// Mitsubishi GX Works2 project: timer   PLC: Q03UDV

PROGRAM MAIN
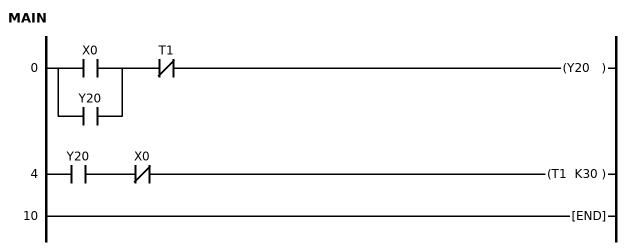
0     LD      X0
      OR      Y20
      ANI     T1
      OUT     Y20
4     LD      Y20
      ANI     X0
      OUT     T1 K30
10    END
END_PROGRAM
